PROGRAM RunGrindingWheel
VAR
END_VAR

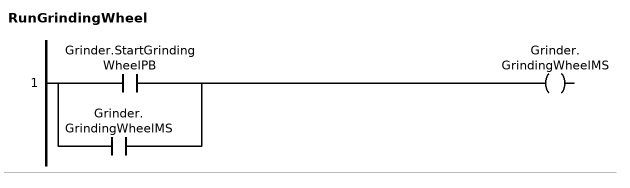
// NETWORK 1
Grinder.GrindingWheelMS := Grinder.StartGrindingWheelPB OR Grinder.GrindingWheelMS;

END_PROGRAM

(* stored: Version 1.1.0.1, ProductVersion 3.1.4024.4
   POU RunGrindingWheel: Id {b3a9820d-1e53-4a7e-9861-db4eac5bf07b}, SpecialFunc None *)
